{library PUBLIC}
(* This function will return the checksum for a specific DataGram message.
  Note: the DataGram is not changed including the CheckSum member by this function, only calculated.
  You need to set the correct value in the DataGram.*)
FUNCTION DatagramCheckSum : BYTE
VAR_INPUT
	Data:		DataGram;
END_VAR
VAR
	Ptr: 		POINTER TO BYTE;
	Size: 		INT;
	i: 			INT;
	CkSum: 	BYTE;
END_VAR

Size:=_DataGramSize()-1;

CkSum:=0;
Ptr:=ADR(Data);

FOR i:=1 TO Size DO
	CkSum:=CkSum+Ptr^;
	Ptr:=Ptr+1;
END_FOR;

DatagramCheckSum:=CkSum;

END_FUNCTION

(* stored: Version 1.1.0.1, ProductVersion 3.1.4022.12
   POU DatagramCheckSum: Id {bfe0295c-f97d-4e83-997b-c956cb80b0bd}, SpecialFunc None *)
